FUNCTION_BLOCK FB_SetPointGenerator
VAR_INPUT
	u : LREAL := 0.0;
	u_t : LREAL := 0.0;
	u_tt : LREAL := 0.0;
END_VAR
VAR_OUTPUT
END_VAR
VAR
	omega : LREAL := 1.0;
	beta : LREAL := 1.0;
	
	Ts : LREAL := 0.005;
	y : LREAL := 0.0;
	y_t : LREAL := 0.0;
	y_tt : LREAL := 0.0;
END_VAR


y_tt := u_tt + 2*beta*omega*(u_t - y_t) + omega*omega*(u - y);
    
y_t := y_t + y_tt*Ts;
    
y := y + y_t*Ts;

METHOD Reset : BOOL
VAR_INPUT
END_VAR
u := 0.0;
u_t := 0.0;
u_tt := 0.0;

y := 0.0;
y_t := 0.0;
y_tt := 0.0;
END_METHOD

METHOD SetBeta : BOOL
VAR_INPUT
	value : LREAL;
END_VAR
beta := ABS(value);
END_METHOD

METHOD SetOmega : BOOL
VAR_INPUT
	value : LREAL;
END_VAR
omega := ABS(value);
END_METHOD

METHOD SetTimeStep : BOOL
VAR_INPUT
	timestep : LREAL;
END_VAR
Ts := ABS(timestep);
END_METHOD

END_FUNCTION_BLOCK

(* stored: Version 1.1.0.1, ProductVersion 3.1.4022.7
   POU FB_SetPointGenerator: Id {fe9902f6-37f1-401e-addb-5933c990711a}, SpecialFunc None
   Method Reset: Id {eca57de5-bf7d-4705-8f61-c9fd3597f754}
   Method SetBeta: Id {054e8021-3bfc-44f4-b38f-da5266ddd1b2}
   Method SetOmega: Id {b817e9a5-d548-431d-b2b3-33fae8ac5011}
   Method SetTimeStep: Id {69aaf3fa-9678-4122-8cc1-cc0182620768} *)
